FUNCTION_BLOCK FB_ExhaustSystemPrint
VAR_INPUT
  bI_FUReady                         AT %I* : BOOL;   (*FU ready*)
  iI_VacuumMeasurement               AT %I* : UINT;   (*Analog input: vacuum measurement*)
  bPrintActive                              : BOOL;   (*Printing active*)
END_VAR

VAR_OUTPUT
  bO_FUActivate                      AT %Q* : BOOL;   (*FU activation*)
  OnExhaustSetpoint                  AT %Q* : UINT;   (*Analog output: pump setpoint*)

  bExhaustError                             : BOOL;   (*Exhaust system ok and ready*)
  // detailed status (for messages)
  bFUReady                                  : BOOL;   (*FU ready*)
  bVacuumWarningLevel                       : BOOL;   (*Vacuum warning level reached*)
  bVacuumErrorLevel                         : BOOL;   (*Vacuum error level reached*)
END_VAR

VAR
  iL_Counter                                : INT;    (*Basic counter*)
  bMappingChecked                           : BOOL;   (*Checked mapped variable status*)
  bMapping_FUReady_Done                     : BOOL;   (*FUReady is mapped*)
  
  fb_TofFUOffDelay                          : TOF;    (*FU off delay*)
  fb_TonVacuumCheckDelay                    : TON;    (*Vacuum check delay*)

  fL_VacuumAnalogLevelMBar                  : REAL;   (*Actual value analog-input in mBar*)
END_VAR

VAR PERSISTENT
  tR_FUOffDelay                             : TIME := T#3M;   (*FU off delay time*)
  tR_VacuumCheckDelay                       : TIME := T#10S;  (*Vacuum check delay time*)

  iR_VacuumAnalogMinDigit                   : UINT := 0;      (*Min value analog-input in digit*)
  iR_VacuumAnalogMaxDigit                   : UINT := 32767;  (*Max value analog-input in digit*)
  fR_VacuumAnalogMinMBar                    : REAL := 0;      (*Min value analog-input in mBar*)
  fR_VacuumAnalogMaxMBar                    : REAL := 50.0;   (*Max value analog-input in mBar*)
  fR_VacuumWarningLevelMBar                 : REAL := 20.0;   (*Warning level in mBar*)
  fR_VacuumErrorLevelMBar                   : REAL := 10.0;   (*Error level in mBar*)

  iR_VacuumPumpSetPercent                   : UINT := 0;      (*Pump setpoinr [%]*)
  iR_VacuumPumpSetpointMaxDigit             : UINT := 13762;  (*Max value analog-output in digit, max pump = 4.2V*)
END_VAR

// mapping check
IF NOT bMappingChecked THEN checkMapping(); END_IF
IF NOT bMapping_FUReady_Done THEN bI_FUReady := TRUE; END_IF    // if not mapped is ready


bFUReady := bI_FUReady;  // AND bO_FUActivate?

fb_TofFUOffDelay(IN := bPrintActive, PT := tR_FUOffDelay);    // turn-off delay
bO_FUActivate := fb_TofFUOffDelay.Q;

fL_VacuumAnalogLevelMBar := UINT_TO_REAL(iI_VacuumMeasurement) * fR_VacuumAnalogMaxMBar / iR_VacuumAnalogMaxDigit;

fb_TonVacuumCheckDelay(IN := bO_FUActivate, PT := tR_VacuumCheckDelay);   // delay for vacum measurement
IF fb_TonVacuumCheckDelay.Q THEN
  // check levels and set waring/error
  bVacuumWarningLevel := fL_VacuumAnalogLevelMBar < fR_VacuumWarningLevelMBar;
  bVacuumErrorLevel   := fL_VacuumAnalogLevelMBar < fR_VacuumErrorLevelMBar;
END_IF


bExhaustError := NOT bFUReady OR (bVacuumErrorLevel AND bO_FUActivate);

OnExhaustSetpoint := REAL_TO_UINT(UINT_TO_REAL(iR_VacuumPumpSetpointMaxDigit) / 100 * iR_VacuumPumpSetPercent);

METHOD PRIVATE checkMapping
VAR_INPUT
END_VAR
bMapping_FUReady_Done := F_GetMappingStatus(p:=ADR(bI_FUReady), n:=SIZEOF(bI_FUReady)) > EPlcMappingStatus.MS_Unmapped;

bMappingChecked := TRUE;
END_METHOD

METHOD mAckError : BOOL
VAR_INPUT
END_VAR
bVacuumWarningLevel := FALSE;
bVacuumErrorLevel   := FALSE;
END_METHOD

END_FUNCTION_BLOCK

(* stored: Version 1.1.0.1, ProductVersion 3.1.4024.11
   POU FB_ExhaustSystemPrint: Id {9d3ade69-02c3-47ed-bd02-3517b9357a0c}, SpecialFunc None
   Method checkMapping: Id {cc586209-65da-4391-8b61-ef801610bd07}
   Method mAckError: Id {f16ec73d-1c7a-41ac-bd19-106bc5fe0258} *)
